// TIA Portal V20 export
// export: Created 2025-12-01T14:57:22.2302247Z, ExportSetting None, DisplayName Totally Integrated Automation Portal, DisplayVersion V20 Update 3, DisplayName TIA Portal Openness, DisplayVersion V20 Update 3, DisplayName TIA Portal Version Control Interface, DisplayVersion V20 Update 3, DisplayName STEP 7 Professional, DisplayVersion V20 Update 3, DisplayName STEP 7 Safety, DisplayVersion V20 Update 2, DisplayName WinCC Basic/Comfort/Advanced, DisplayVersion V20 Update 3, DisplayName WinCC Professional, DisplayVersion V20 Update 3, DisplayName WinCC Unified, DisplayVersion V20 Update 3
DATA_BLOCK "DB908_Sinoptico"   // DB908
{ S7_Optimized_Access := 'FALSE' }
AUTHOR : GENERAL
NAME : 20160415
VERSION : 4.0
// stored: AutoNumber false
   VAR
      Mesa : Array[0.."CTE_MaxMesas"] of Byte;   // 0:Vacia,1:Cargada,2:EnCarga,3:EnDescarga,4:Reset,5,6,7:Error
      MesaCantidadUTs : Array[0.."CTE_MaxMesas"] of Byte;   // 0:Vacia,1:Cargada,2:EnCarga,3:EnDescarga,4:Reset,5,6,7:Error
      ArmarioPotencia : Array[0..5] of Struct   // 0:Vacia,1:Cargada,2:EnCarga,3:EnDescarga,4:Reset,5,6,7:Error
         Linea { S7_SetPoint := 'True'} : Array[0..50] of "UDT_HMI_LineaPotencia";
      END_STRUCT;
      Seta : Array[0..99] of Bool;
      BarreraQ : Array[0..99] of Bool;
      Barrera_Señales { S7_SetPoint := 'True'} : Array[0..99] of "UDT_HMI_SeñalesBarreras";
      Barrera_DIAG : Array[0..99] of Word;
      Galibo_NOOK : Array[0..29] of Bool;
      Galibo_Señal { S7_SetPoint := 'True'} : Array[0..29] of "UDT_HMI_SeñalesGalibo";
      Galibo_Codigo : Array[0..29] of Word;
      Galibo_TacoHueco : Array[0..29] of Word;
      OffsetCCPIF : UInt;
   END_VAR
BEGIN
END_DATA_BLOCK
